TYPE ST_Parameters :
STRUCT
	fCyclicTime : LREAL := 0.01; //[s]
	fMaxVelocityLimit : LREAL := 0.05; //[m/s]
	fBoreArea : LREAL := 0.0033183;
	fAnnulusArea : LREAL := 0.0023562;
	fMaxFlowCapacity : LREAL := 30; //[l/min]
END_STRUCT
END_TYPE

(* stored: Version 1.1.0.1, ProductVersion 3.1.4024.10
   DUT ST_Parameters: Id {28c89b95-688c-4db5-a51b-ee26f2081432} *)
